{attribute addProperty BoxType "EP2816-0003-0016"}
{attribute addProperty Id "DIG_Diag_Inputs_ChannelAT %I*ARRAY[0..8] OF DIG_Diag_Inputs_Channel_AC4A9AF0128160DIG_Inputs_DeviceAT %I*DIG_Inputs_Device_30BACB404050DIG_Output_ChannelAT %Q*ARRAY[0..8] OF DIG_Output_Channel_33B76376128160DIG_Outputs_DeviceAT %Q*DIG_Outputs_Device_735003021620WcStateAT %I*WcState_98A4DF7520.250InfoDataAT %I*InfoData_BC63D37F80100"}
{attribute addProperty CRC "2416013832"}
{attribute addProperty SizeInBites "394"}
{attribute addProperty SizeInBytes "49.25"}
TYPE EP2816_E74B64DB :
STRUCT
	{attribute addProperty Name "DIG_Diag_Inputs_Channel"}
	DIG_Diag_Inputs_Channel : ARRAY[0..8] OF DIG_Diag_Inputs_Channel_AC4A9AF0;
	{attribute addProperty Name "DIG_Inputs_Device"}
	DIG_Inputs_Device : DIG_Inputs_Device_30BACB40;
	{attribute addProperty Name "DIG_Output_Channel"}
	DIG_Output_Channel : ARRAY[0..8] OF DIG_Output_Channel_33B76376;
	{attribute addProperty Name "DIG_Outputs_Device"}
	DIG_Outputs_Device : DIG_Outputs_Device_73500302;
	{attribute addProperty Name "WcState"}
	WcState : WcState_98A4DF75;
	{attribute addProperty Name "InfoData"}
	InfoData : InfoData_BC63D37F;
END_STRUCT
END_TYPE

(* stored: Version 1.2.0.0, ProductVersion 3.1.4024.9
   DUT EP2816_E74B64DB: Id {5cfaa082-6274-49b2-8a72-48f268ce5ef9} *)
